INTERFACE I_Alarms

METHOD PUBLIC Accept
VAR_INPUT
	Visitor : I_AlarmVisitor;
END_VAR
END_METHOD

METHOD AddAlarm
VAR_INPUT
	Alarm : I_Alarm;
END_VAR
END_METHOD

PROPERTY PUBLIC HasRaisedAlarm : BOOL
GET
END_GET
END_PROPERTY

END_INTERFACE

(* stored: Version 1.1.0.1, ProductVersion 3.1.4024.12
   Itf I_Alarms: Id {de85c531-bf50-4dff-8f3c-8b858df680d9}
   Method Accept: Id {a60a68c8-549d-4278-979e-b0c345847604}
   Method AddAlarm: Id {7bf07649-ae5a-4189-924a-ecec0ca95342}
   Property HasRaisedAlarm: Id {dbe30b3a-306f-439d-9c23-64761c18e3a5}
   Get Get: Id {e690e846-ab4c-4f3f-b6f0-5c00ac630b52} *)
